INTERFACE I_PendingResponseManagerConfig

METHOD PUBLIC TryGetResponseIdFromRequest : BOOL
VAR_INPUT
	Request : I_Request;
	Destination : ANY;
END_VAR
END_METHOD

METHOD PUBLIC TryGetSessionIdFromRequest : BOOL
VAR_INPUT
	Request : I_Request;
	Destination : REFERENCE TO T_MAXSTRING;
END_VAR
END_METHOD

END_INTERFACE

(* stored: Version 1.1.0.1, ProductVersion 3.1.4024.12
   Itf I_PendingResponseManagerConfig: Id {17303ec9-1bec-4a17-ab1f-fe3910f2ac30}
   Method TryGetResponseIdFromRequest: Id {207b7440-4700-4749-a52a-b0c85f5c5d69}
   Method TryGetSessionIdFromRequest: Id {73fa9195-0a80-486b-9b7e-5f5e0fe3460c} *)
